TEXTLIST TXT_LIST_PNEMATIC_ACTOR
  1 = 'Timeout: Bewegung nach Arbeitsstellung' | de: 'Timeout: Bewegung nach Arbeitsstellung' | en: 'Timeout: Move to Workposition'
  2 = 'Timeout: Bewegung nach Grundstellung' | de: 'Timeout: Bewegung nach Grundstellung' | en: 'Timeout: Move to Basepostion'
  3 = 'fährt in Grundposition' | de: 'fährt in Grundposition' | en: 'moves to Baseposition'
  4 = 'ist in Grundposition' | de: 'ist in Grundposition' | en: 'in Baseposition'
  5 = 'fährt in Arbeitsposition' | de: 'fährt in Arbeitsposition' | en: 'moves to Workposition'
  6 = 'ist in Arbeitsposition' | de: 'ist in Arbeitsposition' | en: 'in Workposition'
  7 = 'in undefinierter Position' | de: 'in undefinierter Position' | en: 'in undefined postion'
  8 = 'Timeout bei Fahrt nach Grundstellung' | de: 'Timeout bei Fahrt nach Grundstellung' | en: 'Timeout: Move to Basepos.'
  9 = 'Timeout bei Fahrt nach Arbeitsstellung' | de: 'Timeout bei Fahrt nach Arbeitsstellung' | en: 'Timeout: Move to Workpos.'
  11 = 'Vakuum ein / Druck nicht erreicht' | de: 'Vakuum ein / Druck nicht erreicht' | en: 'vaccum on / pressure NOK'
  12 = 'Vakuum ein / Druck OK' | de: 'Vakuum ein / Druck OK' | en: 'vaccum on / pressure OK'
  13 = 'Abblasen ein' | de: 'Abblasen ein' | en: 'blow out'
  14 = 'nicht aktiv' | de: 'nicht aktiv' | en: 'not active'
  15 = 'ist in Mittelstellung' | de: 'ist in Mittelstellung' | en: 'in mid position'
  16 = 'blockiert durch' | de: 'blockiert durch' | en: 'locked by'
   = ''
END_TEXTLIST

(* stored: Version 1.1.0.1, ProductVersion 3.1.4024.12
   TextList TXT_LIST_PNEMATIC_ACTOR: Id {8c9f483a-8540-47eb-89f4-d680911906ae} *)
